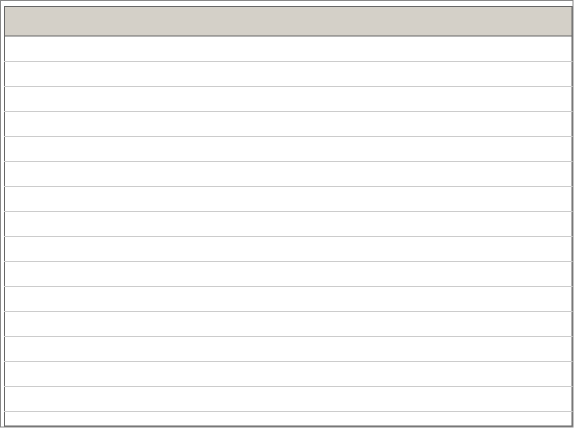
VISUALIZATION Err_record  // 574x428
    Table (4,6 568x420), data array: Error_List
        p3854506369: Error_List[INDEX].Timer
        p1892666644: Error_List[INDEX].Axis
        p338671338: Error_List[INDEX].ErrorID
        p2170511999: Error_List[INDEX].ErrorTXT
        p3723444502: Error_List[INDEX].ErrorCNT
END_VISUALIZATION

(* stored: Version 1.1.0.1, ProductVersion 3.1.4018.5
   Visu Err_record: Id {8fdcf082-8165-4b4f-916b-9e3d80297abd} *)
